# EPICS substitutions: iocs/cpscExample/iocBoot/ioccpscExample/cpsc.substitutions
file "$(MOTOR)/db/asyn_motor.db"
{
pattern
{ M,         DTYP,   PORT,  ADDR,       DESC,  EGU,  DIR,  VMAX,  VELO,  VBAS,  ACCL,  BDST,  BVEL,  BACC,   MRES,  PREC,  DHLM,  DLLM,  INIT}
{m1,  "asynMotor",  CPSC1,     0,  "Motor 1",   um,  Pos,  15.0,   3.0,  0.05,   0.5,     0,   1.0,     2,  0.001,     9,     0,     0,    ""}
{m2,  "asynMotor",  CPSC1,     1,  "Motor 2",   um,  Pos,  15.0,   3.0,  0.05,   0.5,     0,   1.0,     2,  0.001,     9,     0,     0,    ""}
{m3,  "asynMotor",  CPSC1,     2,  "Motor 3",   um,  Pos,  15.0,   3.0,  0.05,   0.5,     0,   1.0,     2,  0.001,     9,     0,     0,    ""}
}
